Staubli VAL3: USERPAGE.dtx

bool Show
public bool bListItemRef
bool bReadWrite = true
public bool bShowDialog
public bool bUseEscape
public bool bUseRefresh = true
public num nBottomX[2]
  [0] = 18
  [1] = 18
public num nBottomY = 11
num nFirst
num nKey
num nOffSet
num nOldValue[2]
  [0] = 200
  [1] = 200
public num nPage = 100000
public num nParaAdjustType
num nTest
public num nToSuperV = -1
public num nTopX[2]
  [0] = 20
  [1] = 20
public num nTopY
public num nView
public string sItems = "Name"
string sMessage = "是否删除该项?"
public string sTitle = "工具"
public string sToSuperV
string stest[11]
  [0] = "sbx"
  [1] = "sdfgsd"
  [2] = "bsfghsfh"
  [3] = "sdfgsdfg"
  [4] = "shsgh"
  [5] = "ghdfh"
  [6] = "snsfg"
  [7] = "sfgsg"
  [8] = "sfgsdfg"
  [9] = "sfgs"
  [10] = "dfsgs"
string stest2
string stest3
